// TIA Portal V20 export
TYPE "typeFDoorFunctionData"
// Safety status of door
// stored: Access Published, IsFailsafeCompliant true, Namespace Safety
   STRUCT
      STO : Bool;   // STO, safet torque of for drives
      released { ExternalWritable := 'False'} : Bool;   // Door Locked, Reset Done
      ackReq { ExternalWritable := 'False'} : Bool;   // Acknowledge required
   END_STRUCT;
END_TYPE
